Yaskawa INFORM job: R2_W37-38-A2(90,0)_MP_OK.JBI

/JOB
//NAME R2_W37-38-A2(90,0)_MP_OK
///FOLDERNAME MP_TEST
//POS
///NPOS 37,37,0,2,0,0
///TOOL 0
///POSTYPE PULSE
///PULSE
C00000=59274,-2798,-33333,-1733,105875,38300
C00001=66056,-40423,-104269,-1733,105875,38300
C00002=106246,-40423,-104269,-1733,105875,38300
C00003=153029,-40423,-104269,-1733,105875,38300
C00004=183647,-58567,-106484,-21191,125994,67618
C00005=224116,-16297,-78542,-22423,105508,69475
C00006=210077,-31788,-66157,-45162,73373,64375
C00007=178964,14537,-16406,-30186,55210,57821
C00008=176669,18772,-10786,-29107,53313,57381
C00009=176195,18706,-9766,-29024,52574,57395
C00010=176195,18472,-8428,-29376,51745,57656
C00011=179062,14046,-13909,-30889,53693,58356
C00012=189891,47583,14821,-51298,83276,63796
C00013=189430,45805,12918,-51165,83193,63607
C00014=189891,47583,14821,-51298,83276,63796
C00015=178070,11995,-17162,-29890,54171,57749
C00016=178072,11999,-17154,-29892,54170,57750
C00017=178070,11995,-17162,-29890,54171,57749
C00018=178209,12482,-17565,-29808,54654,57660
C00019=178555,13757,-18519,-29617,55856,57440
C00020=197438,24102,-8473,-62088,77366,-49969
C00021=193120,61905,28460,-57219,91858,-72182
C00022=192302,57705,26606,-57037,90807,-71942
C00023=191968,56074,25940,-56969,90369,-71840
C00024=191964,56191,24825,-56995,90787,-72127
C00025=192675,56292,26177,-57078,90766,-71695
C00026=187770,39139,10168,-54323,74163,-71832
C00027=192147,56758,29144,-56075,75144,-69941
C00028=192373,57859,29205,-56028,75580,-70103
C00029=192931,60718,29502,-55933,76648,-70492
C00030=240126,15837,-22502,-63787,104557,-68393
C00031=210077,-31788,-66157,-45162,73373,64375
C00032=224116,-16297,-78542,-22423,105508,69475
C00033=183647,-58567,-106484,-21191,125994,67618
C00034=153029,-40423,-104269,-1733,105875,38300
C00035=106246,-40423,-104269,-1733,105875,38300
C00036=66056,-40423,-104269,-1733,105875,38300
BC00000=158786,223116,705218
BC00001=158786,223116,705218
BC00002=158786,311299,705218
BC00003=158786,311299,705218
BC00004=350491,216601,295600
BC00005=398174,163325,53
BC00006=398174,163325,53
BC00007=398174,163325,53
BC00008=398174,163325,53
BC00009=398174,163325,53
BC00010=398174,163325,53
BC00011=398174,154203,53
BC00012=398174,149434,53
BC00013=398174,149426,53
BC00014=398174,149434,53
BC00015=398174,152461,53
BC00016=398174,150157,53
BC00017=398174,152461,53
BC00018=398174,155067,53
BC00019=398174,161583,53
BC00020=398174,147870,53
BC00021=398174,140034,53
BC00022=398174,136953,53
BC00023=398174,135721,53
BC00024=398174,135721,53
BC00025=398174,135721,53
BC00026=398174,148637,53
BC00027=398174,128850,53
BC00028=398174,130635,53
BC00029=398174,135097,53
BC00030=398174,135097,53
BC00031=398174,163325,53
BC00032=398174,163325,53
BC00033=350491,216601,295600
BC00034=158786,311299,705218
BC00035=158786,311299,705218
BC00036=158786,223116,705218
///POSTYPE BASE
///RECTAN
///RCONF 0,0,0,0,0,0,0,0,0,0,0,0,0,0,0,0,0,0,0,0,0,0,0,0
P00006=0.222,-3.123,-1.508,0.0000,0.0000,0.0000
P00023=0.143,-0.036,0.682,0.0000,0.0000,0.0000
//INST
///DATE 2023/11/16 10:46
///ATTR SC,RW
///GROUP1 RB1,BS1
NOP
'r2_W37-38-A2(90,0)
'Path S953
MOVJ C00000 BC00000 VJ=20.00
MOVJ C00001 BC00001 VJ=20.00
MOVJ C00002 BC00002 VJ=20.00
MOVJ C00003 BC00003 VJ=20.00
MOVJ C00004 BC00004 VJ=20.00
MOVJ C00005 BC00005 VJ=20.00
MOVJ C00006 BC00006 VJ=20.00
SFTOF
MOVJ C00007 BC00007 VJ=20.00
MOVL C00008 BC00008 V=100.0
MOVL C00009 BC00009 V=60.0
REFP 3 C00010 BC00010
CALL JOB:SEARCH-R1
SET P023 P006
SFTON P023
MOVL C00011 BC00011 V=60.0
MOVL C00012 BC00012 V=60.0
REFP 3 C00013 BC00013
CALL JOB:SEARCH-R1
SET P023 P006
SFTON P023
MOVL C00014 BC00014 V=60.0
MOVL C00015 BC00015 V=60.0
REFP 3 C00016 BC00016
CALL JOB:SEARCH-R1
SET P023 P006
SFTON P023
MOVL C00017 BC00017 V=60.0
MOVL C00018 BC00018 V=100.0
MOVL C00019 BC00019 V=100.0
'Path VIA955
SFTOF
MOVJ C00020 BC00020 VJ=20.00
'Path W954
SFTOF
SFTON P023
MOVJ C00021 BC00021 VJ=20.00
MOVL C00022 BC00022 V=100.0
MACRO1 MJ#(0) ARGF8
MOVL C00023 BC00023 V=100.0 PL=0
REFP 1 C00024 BC00024
REFP 2 C00025 BC00025
ARCON
MOVL C00026 BC00026 V=10.0
MOVL C00027 BC00027 V=10.0
ARCOF
MOVL C00028 BC00028 V=100.0
MOVL C00029 BC00029 V=100.0
SFTOF
MOVJ C00030 BC00030 VJ=20.00
MOVJ C00031 BC00031 VJ=20.00
MOVJ C00032 BC00032 VJ=20.00
MOVJ C00033 BC00033 VJ=20.00
MOVJ C00034 BC00034 VJ=20.00
MOVJ C00035 BC00035 VJ=20.00
MOVJ C00036 BC00036 VJ=20.00
'
END
